FUNCTION_BLOCK AR_CALIBRATE_SQ (* Adapter-based sequential two-point calibration (offset then scale) with ECC-enforced order *)
  (* Standard: 61499-1 *)
  (* Version 1.0, 2026-06-01, Meisterschulen am Ostbahnhof *)
  PACKAGE adapter::Engineering::measurements;
  (* Documentation:
  Formula
    Y = (X + OFFSET) * SCALE Calibration (Two-Point, ECC-Enforced)
    - Offset (CO): Apply low reference, set Y_Offset to desired output, trigger CO
   OFFSET := Y_Offset / SCALE - X → after CO, Y always equals Y_Offset (independent of SCALE)
   - Scale (CS): Apply high reference, set Y_Scale to desired output, trigger CS
   Calculates SCALE and OFFSET decoupled using both reference points → after CS, the line passes exactly through both points
    Note: Both Y_Offset and Y_Scale are target values on the output side.
    - CS is only reachable after offset calibration (state WAIT_CS) – enforced by ECC
   - CO can be repeated at any time to re-calibrate offset
   - Normal calculation via X.E1 works in all states
    Key Difference vs. AR_CALIBRATE
      Feature |  AR_CALIBRATE |  AR_CALIBRATE_SQ |  
    CO formula |  OFFSET := Y_Offset - X |  OFFSET := Y_Offset / SCALE - X |  
    Y after CO |  Y = Y_Offset * SCALE
   (only correct when SCALE = 1) |  Y = Y_Offset
   (always correct) |  
    Order enforcement |  None (both directly accessible) |  ECC-enforced (CO before CS) |
  *)
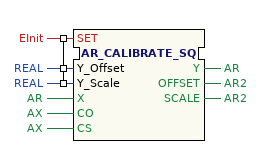
  EVENT_INPUT
    SET : EInit WITH Y_Offset, Y_Scale; (* Set References *)
  END_EVENT
  VAR_INPUT
    Y_Offset : REAL; (* Target output Y at low calibration point (offset) *)
    Y_Scale : REAL; (* Target output Y at high calibration point (scale) *)
  END_VAR
  SOCKETS
    X : adapter::types::unidirectional::AR; (* Raw Input *)
    CO : adapter::types::unidirectional::AX; (* Calibrate Offset *)
    CS : adapter::types::unidirectional::AX; (* Calibrate Scale *)
  END_SOCKETS
  PLUGS
    Y : adapter::types::unidirectional::AR; (* Calibrated Output *)
    OFFSET : adapter::types::bidirectional::AR2; (* Stored offset value (initial 0.0) *)
    SCALE : adapter::types::bidirectional::AR2; (* Stored scale value (initial 1.0) *)
  END_PLUGS
  VAR
    X_LOW_INT : REAL; (* Stored raw value at CO *)
    Y_LOW_INT : REAL; (* Stored target value at CO *)
  END_VAR
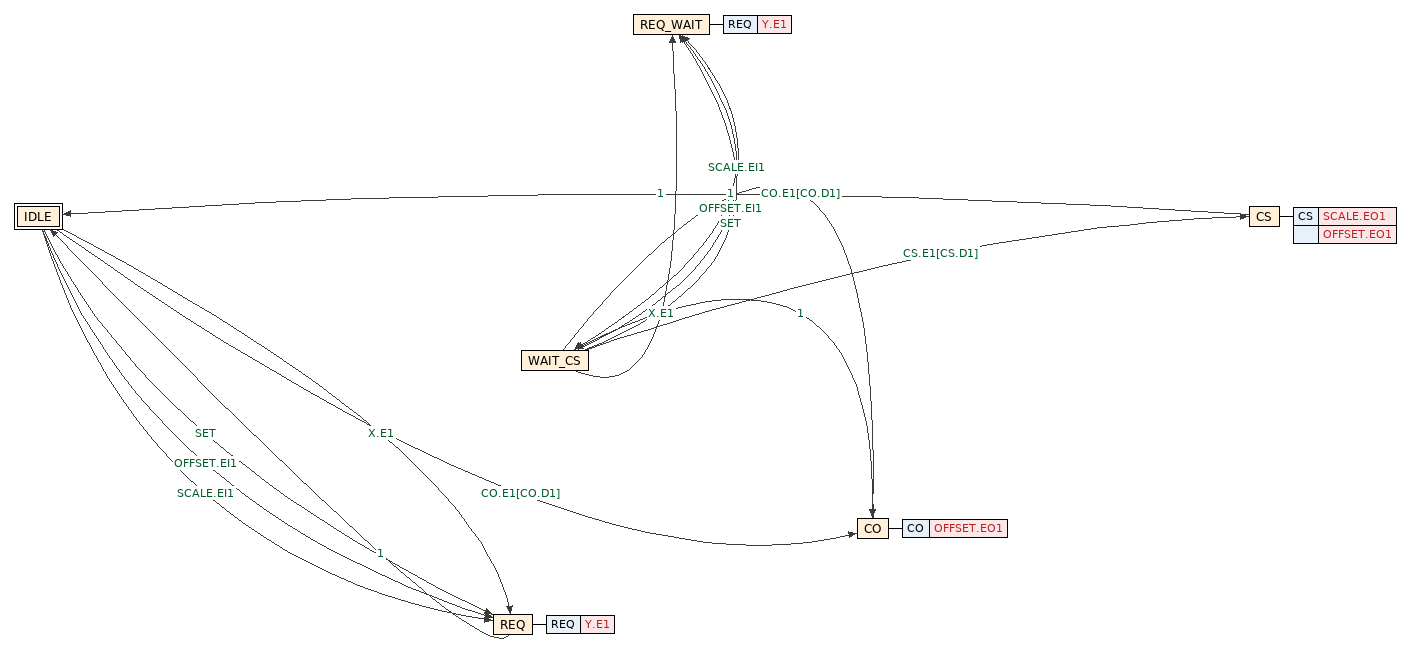
  EC_STATES
    IDLE;
    REQ : REQ -> Y.E1;
    CO : CO -> OFFSET.EO1;
    WAIT_CS;
    REQ_WAIT : REQ -> Y.E1;
    CS : CS -> SCALE.EO1, -> OFFSET.EO1;
  END_STATES
  EC_TRANSITIONS
    IDLE TO REQ := X.E1;
    REQ TO IDLE := 1;
    IDLE TO CO := CO.E1[CO.D1];
    CO TO WAIT_CS := 1;
    WAIT_CS TO REQ_WAIT := X.E1;
    REQ_WAIT TO WAIT_CS := 1;
    WAIT_CS TO CS := CS.E1[CS.D1];
    CS TO IDLE := 1;
    WAIT_CS TO CO := CO.E1[CO.D1];
    IDLE TO REQ := SET;
    IDLE TO REQ := OFFSET.EI1;
    IDLE TO REQ := SCALE.EI1;
    WAIT_CS TO REQ_WAIT := SET;
    WAIT_CS TO REQ_WAIT := OFFSET.EI1;
    WAIT_CS TO REQ_WAIT := SCALE.EI1;
  END_TRANSITIONS
  ALGORITHM REQ IN ST: (* REQ *)
(* calculate calibrated output *)
Y.D1 := (X.D1 + OFFSET.DI1) * SCALE.DI1;
  END_ALGORITHM
  ALGORITHM CO IN ST: (* CO *)
X_LOW_INT := X.D1;
Y_LOW_INT := Y_Offset;
IF SCALE.DI1 <> 0.0 THEN
	OFFSET.DO1 := Y_Offset / SCALE.DI1 - X.D1;
ELSE
	OFFSET.DO1 := Y_Offset - X.D1;
END_IF;
  END_ALGORITHM
  ALGORITHM CS IN ST: (* CS *)
IF (X.D1 - X_LOW_INT) <> 0.0 THEN
	SCALE.DO1 := (Y_Scale - Y_LOW_INT) / (X.D1 - X_LOW_INT);
	IF SCALE.DO1 <> 0.0 THEN
		OFFSET.DO1 := Y_LOW_INT / SCALE.DO1 - X_LOW_INT;
	END_IF;
END_IF;
  END_ALGORITHM
END_FUNCTION_BLOCK
